PROGRAM S1_01_WasherJets_5
VAR
	HMI_Motion: FB_HMI_Control;
	Motion: FB_Motion2way;

	tMessageOffset: UINT;
	tNumMessagesPerRow: UINT;
	
	
	MyAdvanceInterlock: BOOL;
	MyReturnInterlock: BOOL;
	
	MyAutoAdvanceCondition: BOOL;
	MyAutoReturnCondition: BOOL;
	testword: WORD;
	myAdvancePrompt: BOOL;
	myReturnPrompt: BOOL;
	advancedSensor: BOOL;
	returnedSensor: BOOL;
	AdvanceCoil: BOOL;
	ReturnCoil: BOOL;
	tWaitMsgXICAdv: BOOL;
	tWaitMsgXICRet: BOOL;
	FB_SimMotion: FB_SimMotion;
END_VAR

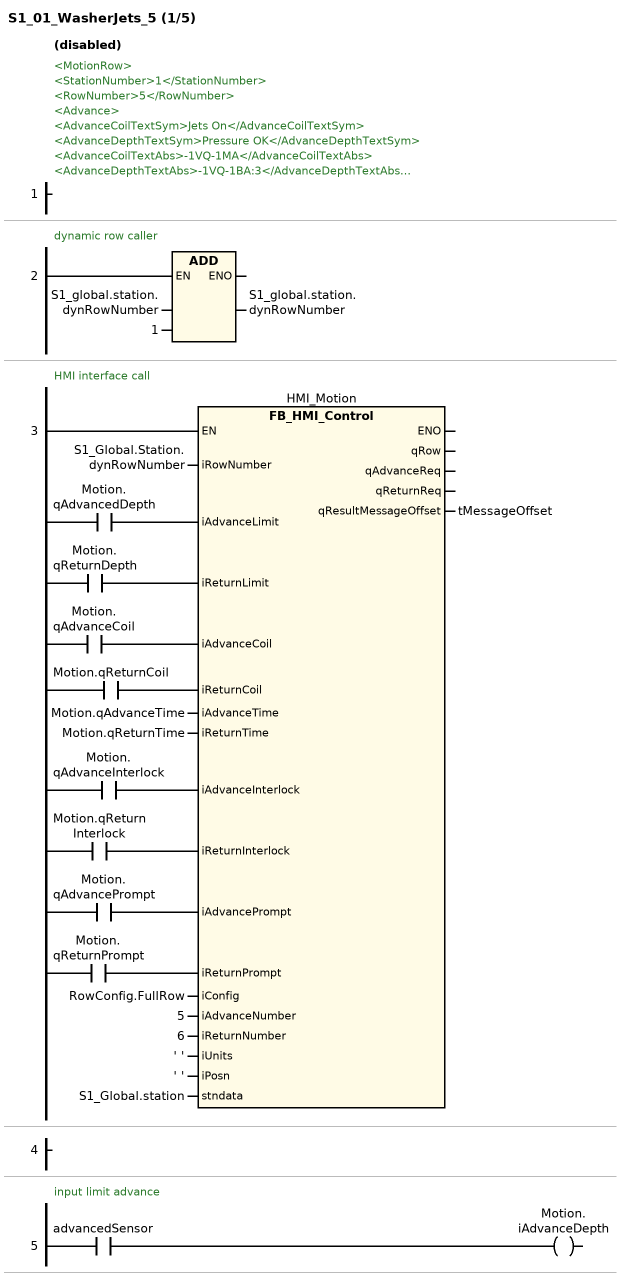
// NETWORK 1 (disabled)
// <MotionRow>
// <StationNumber>1</StationNumber>
// <RowNumber>5</RowNumber>
//   <Advance>
//     <AdvanceCoilTextSym>Jets On</AdvanceCoilTextSym>
//     <AdvanceDepthTextSym>Pressure OK</AdvanceDepthTextSym>
//     <AdvanceCoilTextAbs>-1VQ-1MA</AdvanceCoilTextAbs>
//     <AdvanceDepthTextAbs>-1VQ-1BA:3</AdvanceDepthTextAbs>
//     <ManSeq>5</ManSeq>
//   </Advance>
//   <Return>
//     <ReturnCoilTextSym>Jets Off</ReturnCoilTextSym>
//     <ReturnDepthTextSym>Pressure Off</ReturnDepthTextSym>
//     <ReturnCoilTextAbs>-1VQ-1MA</ReturnCoilTextAbs>
//     <ReturnDepthTextAbs>-1VQ-2BA:3</ReturnDepthTextAbs>
//    <ManSeq>6</ManSeq>
//   </Return>
//   <Motion>
//     <NameSym>Washer Jets</NameSym>
//     <NameAbs>-1VQ</NameAbs>
//   </Motion>
// </MotionRow>

// NETWORK 2
// dynamic row caller
S1_global.station.dynRowNumber := S1_global.station.dynRowNumber + 1;

// NETWORK 3
// HMI interface call
HMI_Motion(
    iRowNumber := S1_Global.Station.dynRowNumber,
    iAdvanceLimit := Motion.qAdvancedDepth,
    iReturnLimit := Motion.qReturnDepth,
    iAdvanceCoil := Motion.qAdvanceCoil,
    iReturnCoil := Motion.qReturnCoil,
    iAdvanceTime := Motion.qAdvanceTime,
    iReturnTime := Motion.qReturnTime,
    iAdvanceInterlock := Motion.qAdvanceInterlock,
    iReturnInterlock := Motion.qReturnInterlock,
    iAdvancePrompt := Motion.qAdvancePrompt,
    iReturnPrompt := Motion.qReturnPrompt,
    iConfig := RowConfig.FullRow,
    iAdvanceNumber := 5,
    iReturnNumber := 6,
    iUnits := ' ',
    iPosn := ' ',
    stndata := S1_Global.station,
    qResultMessageOffset => tMessageOffset); // FB_HMI_Control

// NETWORK 4

// NETWORK 5
// input limit advance
Motion.iAdvanceDepth := advancedSensor;

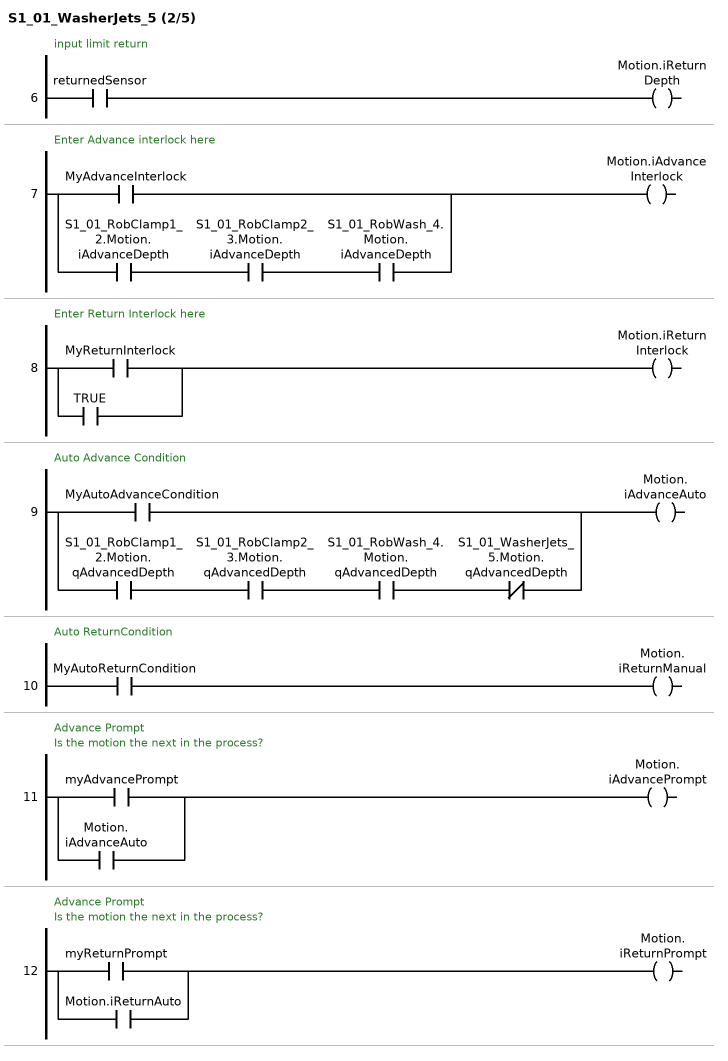
// NETWORK 6
// input limit return
Motion.iReturnDepth := returnedSensor;

// NETWORK 7
// Enter Advance interlock here
Motion.iAdvanceInterlock := MyAdvanceInterlock OR S1_01_RobClamp1_2.Motion.iAdvanceDepth AND S1_01_RobClamp2_3.Motion.iAdvanceDepth AND S1_01_RobWash_4.Motion.iAdvanceDepth;

// NETWORK 8
// Enter Return Interlock here
Motion.iReturnInterlock := MyReturnInterlock OR TRUE;

// NETWORK 9
// Auto Advance Condition
Motion.iAdvanceAuto := MyAutoAdvanceCondition OR S1_01_RobClamp1_2.Motion.qAdvancedDepth AND S1_01_RobClamp2_3.Motion.qAdvancedDepth AND S1_01_RobWash_4.Motion.qAdvancedDepth AND NOT S1_01_WasherJets_5.Motion.qAdvancedDepth;

// NETWORK 10
// Auto ReturnCondition
Motion.iReturnManual := MyAutoReturnCondition;

// NETWORK 11
// Advance Prompt
// Is the motion the next in the process?
Motion.iAdvancePrompt := myAdvancePrompt OR Motion.iAdvanceAuto;

// NETWORK 12
// Advance Prompt
// Is the motion the next in the process?
Motion.iReturnPrompt := myReturnPrompt OR Motion.iReturnAuto;

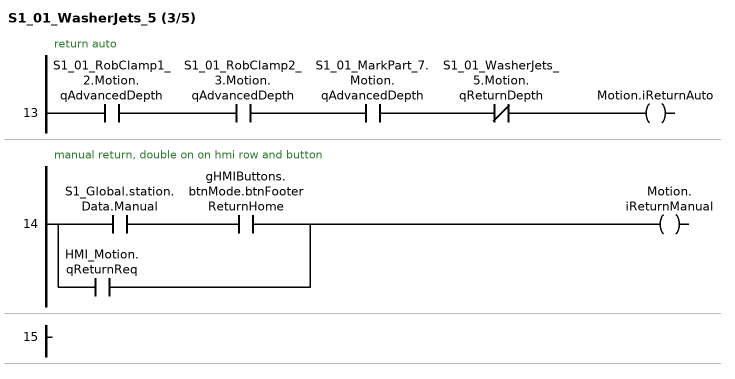
// NETWORK 13
// return auto
Motion.iReturnAuto := S1_01_RobClamp1_2.Motion.qAdvancedDepth AND S1_01_RobClamp2_3.Motion.qAdvancedDepth AND S1_01_MarkPart_7.Motion.qAdvancedDepth AND NOT S1_01_WasherJets_5.Motion.qReturnDepth;

// NETWORK 14
// manual return, double on on hmi row and button
Motion.iReturnManual := S1_Global.station.Data.Manual AND gHMIButtons.btnMode.btnFooterReturnHome OR HMI_Motion.qReturnReq;

// NETWORK 15

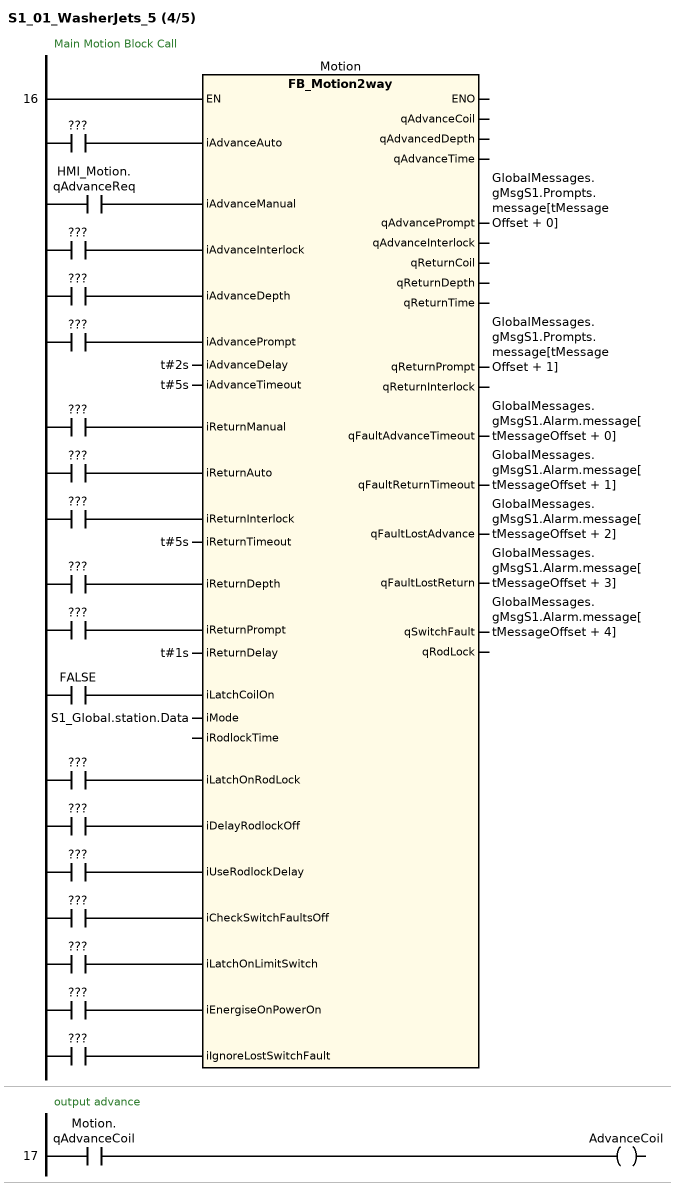
// NETWORK 16
// Main Motion Block Call
Motion(
    iAdvanceManual := HMI_Motion.qAdvanceReq,
    iAdvanceDelay := t#2s,
    iAdvanceTimeout := t#5s,
    iReturnTimeout := t#5s,
    iReturnDelay := t#1s,
    iLatchCoilOn := FALSE,
    iMode := S1_Global.station.Data,
    qAdvancePrompt => GlobalMessages.gMsgS1.Prompts.message[tMessageOffset + 0],
    qReturnPrompt => GlobalMessages.gMsgS1.Prompts.message[tMessageOffset + 1],
    qFaultAdvanceTimeout => GlobalMessages.gMsgS1.Alarm.message[tMessageOffset + 0],
    qFaultReturnTimeout => GlobalMessages.gMsgS1.Alarm.message[tMessageOffset + 1],
    qFaultLostAdvance => GlobalMessages.gMsgS1.Alarm.message[tMessageOffset + 2],
    qFaultLostReturn => GlobalMessages.gMsgS1.Alarm.message[tMessageOffset + 3],
    qSwitchFault => GlobalMessages.gMsgS1.Alarm.message[tMessageOffset + 4]); // FB_Motion2way

// NETWORK 17
// output advance
AdvanceCoil := Motion.qAdvanceCoil;

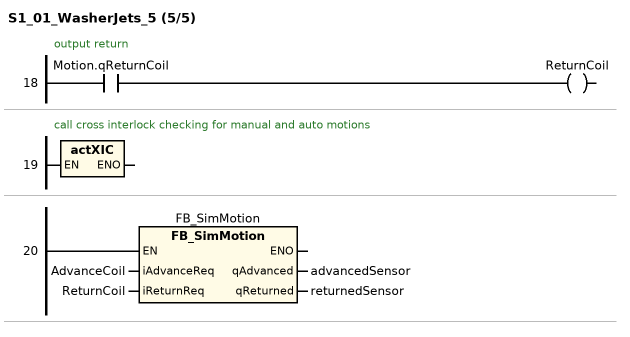
// NETWORK 18
// output return
ReturnCoil := Motion.qReturnCoil;

// NETWORK 19
// call cross interlock checking for manual and auto motions
actXIC();

// NETWORK 20
FB_SimMotion(
    iAdvanceReq := AdvanceCoil,
    iReturnReq := ReturnCoil,
    qAdvanced => advancedSensor,
    qReturned => returnedSensor);

ACTION actXIC:
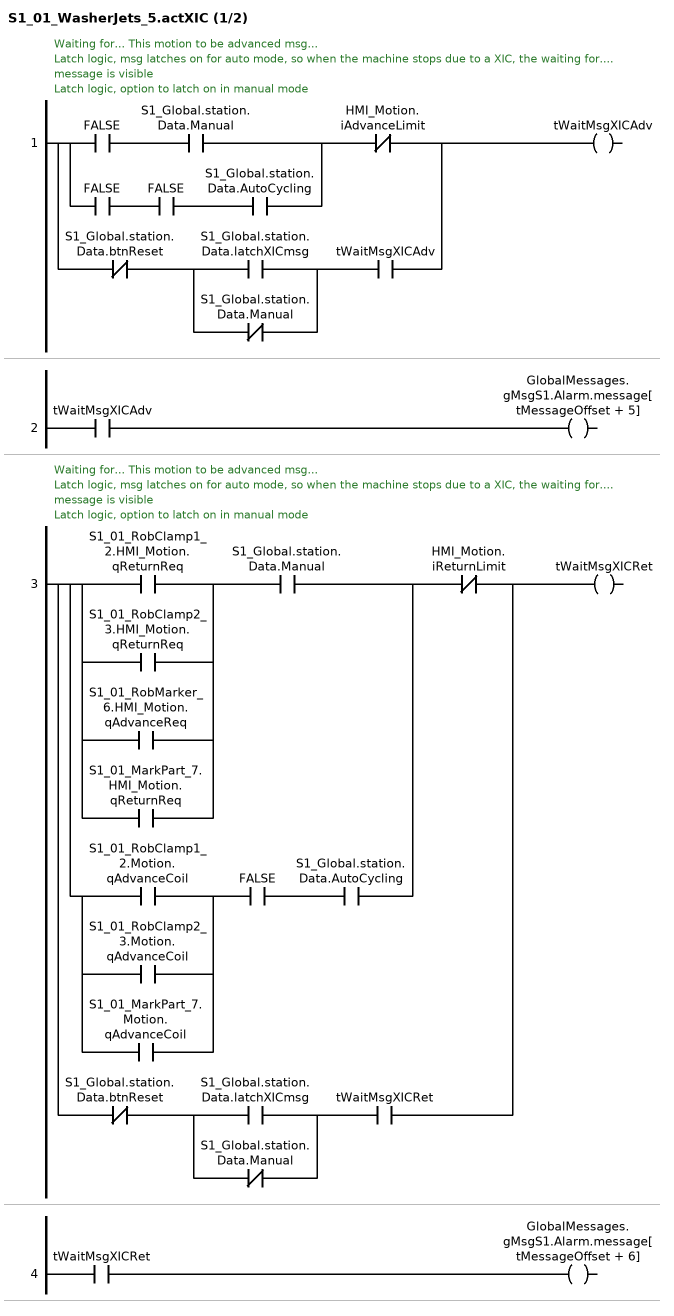
// NETWORK 1
// Waiting for... This motion to be advanced msg...
// Latch logic, msg latches on for auto mode, so when the machine stops due to a XIC, the waiting for.... message is visible
// Latch logic, option to latch on in manual mode
tWaitMsgXICAdv := (FALSE AND S1_Global.station.Data.Manual OR FALSE AND FALSE AND S1_Global.station.Data.AutoCycling) AND NOT HMI_Motion.iAdvanceLimit OR NOT S1_Global.station.Data.btnReset AND (S1_Global.station.Data.latchXICmsg OR NOT S1_Global.station.Data.Manual) AND tWaitMsgXICAdv;

// NETWORK 2
GlobalMessages.gMsgS1.Alarm.message[tMessageOffset + 5] := tWaitMsgXICAdv;

// NETWORK 3
// Waiting for... This motion to be advanced msg...
// Latch logic, msg latches on for auto mode, so when the machine stops due to a XIC, the waiting for.... message is visible
// Latch logic, option to latch on in manual mode
tWaitMsgXICRet := ((S1_01_RobClamp1_2.HMI_Motion.qReturnReq OR S1_01_RobClamp2_3.HMI_Motion.qReturnReq OR S1_01_RobMarker_6.HMI_Motion.qAdvanceReq OR S1_01_MarkPart_7.HMI_Motion.qReturnReq) AND S1_Global.station.Data.Manual OR (S1_01_RobClamp1_2.Motion.qAdvanceCoil OR S1_01_RobClamp2_3.Motion.qAdvanceCoil OR S1_01_MarkPart_7.Motion.qAdvanceCoil) AND FALSE AND S1_Global.station.Data.AutoCycling) AND NOT HMI_Motion.iReturnLimit OR NOT S1_Global.station.Data.btnReset AND (S1_Global.station.Data.latchXICmsg OR NOT S1_Global.station.Data.Manual) AND tWaitMsgXICRet;

// NETWORK 4
GlobalMessages.gMsgS1.Alarm.message[tMessageOffset + 6] := tWaitMsgXICRet;

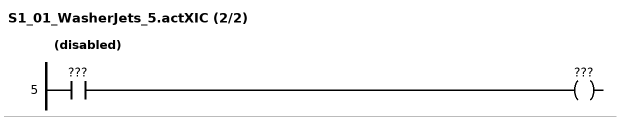
// NETWORK 5 (disabled)
// ??? := ???;
END_ACTION

END_PROGRAM

(* stored: Version 1.1.0.1, ProductVersion 3.1.4024.11
   POU S1_01_WasherJets_5: Id {92d8887f-94ee-43c8-8d41-fae7d953be66}, SpecialFunc None
   Action actXIC: Id {70cdeea7-8270-0340-103b-b49fa02498b8} *)
